{attribute addProperty BoxType "EJ7031-0000-0026"}
{attribute addProperty Id "EnableBIT10.1251ResetBIT10.1252Reduce_torqueBIT10.1253"}
{attribute addProperty CRC "427523686"}
{attribute addProperty SizeInBites "16"}
{attribute addProperty SizeInBytes "2"}
TYPE Control_197B7E66 :
STRUCT
	{attribute addProperty Name "Enable"}
	Enable : BOOL;
	{attribute addProperty Name "Reset"}
	Reset : BOOL;
	{attribute addProperty Name "Reduce_torque"}
	Reduce_torque : BOOL;
	{attribute 'hide'}
	reserve_1_BIT_0 : BOOL;
	{attribute 'hide'}
	reserve_1_BIT_1 : BOOL;
	{attribute 'hide'}
	reserve_1_BIT_2 : BOOL;
	{attribute 'hide'}
	reserve_1_BIT_3 : BOOL;
	{attribute 'hide'}
	reserve_1_BIT_4 : BOOL;
	{attribute 'hide'}
	reserve_2 : BYTE;
END_STRUCT
END_TYPE

(* stored: Version 1.2.0.0, ProductVersion 3.1.4024.9
   DUT Control_197B7E66: Id {bb74c827-4ae8-481f-b8ab-5a7ed64da27e} *)
